FUNCTION_BLOCK FB_Cylinder_DualPWM_SingleSensor EXTENDS FB_Cylinder_SingleSensor
VAR_INPUT
END_VAR
VAR_OUTPUT
END_VAR
VAR
	fbPWMControl		: FB_Enfield_LSV_PWM_SolenoidControl;
	
	//Internal Property Values
	nDutyCycle		: INT := 100;
	
END_VAR

PROPERTY DutyCycle : INT
GET
DutyCycle := nDutyCycle;
END_GET
SET
nDutyCycle := DutyCycle;
END_SET
END_PROPERTY

METHOD HardwareUpdate : BOOL
VAR_INPUT
END_VAR
SUPER^.HardwareUpdate();

IF bExtendCommand THEN
	fbPWMControl.Actuate(nDutyCycle);
ELSIF bRetractCommand THEN
	fbPWMControl.Actuate(nDutyCycle * -1);
ELSE
	fbPWMControl.Actuate(0);
END_IF
END_METHOD

METHOD Monitoring : BOOL
VAR_INPUT
END_VAR
SUPER^.Monitoring();

bReady := bEnabled AND fbPWMControl.Ready AND NOT bError;
END_METHOD

END_FUNCTION_BLOCK

(* stored: Version 1.1.0.1, ProductVersion 3.1.4024.9
   POU FB_Cylinder_DualPWM_SingleSensor: Id {318db1bc-0a06-4ffb-9012-89daaeb9bc1a}, SpecialFunc None
   Folder 01_SUPER_Overrides: Id {4e9aac27-b4d0-45e9-a8ea-d8d2774b9a5b}
   Property DutyCycle: Id {c6923355-0b5c-46d9-9040-4816adac8472}
   Get Get: Id {f3b32ca2-9196-4022-8cf5-d9cef53d120e}
   Set Set: Id {3773468b-66dc-46d2-8138-4fdc549dff54}
   Method HardwareUpdate: Id {1ffcfdb0-8ea4-4d67-a206-52db57326b17}
   Method Monitoring: Id {eb888dc5-8060-405e-9727-c4602ba1f168} *)
